(* Logix 5000 project; controller VET 1756-L62 rev 19.52; software revision 19.01; part 24 of 27 *)
(* tags used below, declared in another part *)
   Automatismos : DINT;
   Aux : DINT[500];
   EColor : DINT[1000];
   Eqp : Equipo[50];
   Errors : Fault_Register;
   I : Index;
   RunStarts : DINT[1000];
   String : STRING[40];
   TabEqp : INT[500];
   _Codes : DINT[500];
   _Eqp : Equipo[800];
   _Eqp_Cfg : Eqp_Cfg[800];
   _Origen : Origen[40];
   _Parametros_F : REAL[30];
   _SS : Soft_Starter[20];
   _Typlgie : Eqp_Typologie[800];   // Process Flow Typologie
   Batch : batch[10];
   borrar : DINT[100];
   corriente : REAL[40];
   fecha_plc : DINT;
   flujometro : flujometro[5];
   hora_plc : DINT;
   peso_tolva : REAL[80];
   Set_Global : DINT[20];
   SetDInt : DINT[500];
   simulacion : BOOL;
   SS_Comun : Soft_Starter;
   SSvar : set_variables;
   TabBin : Bins_Setup;
   Timer : TIMER[500];
   Value : DINT[500];
   vdf : VDFS[20];
   VDFidx : DINT;
(* Main1, continued *)

ROUTINE _Cntrl_Valve   (* ladder *)
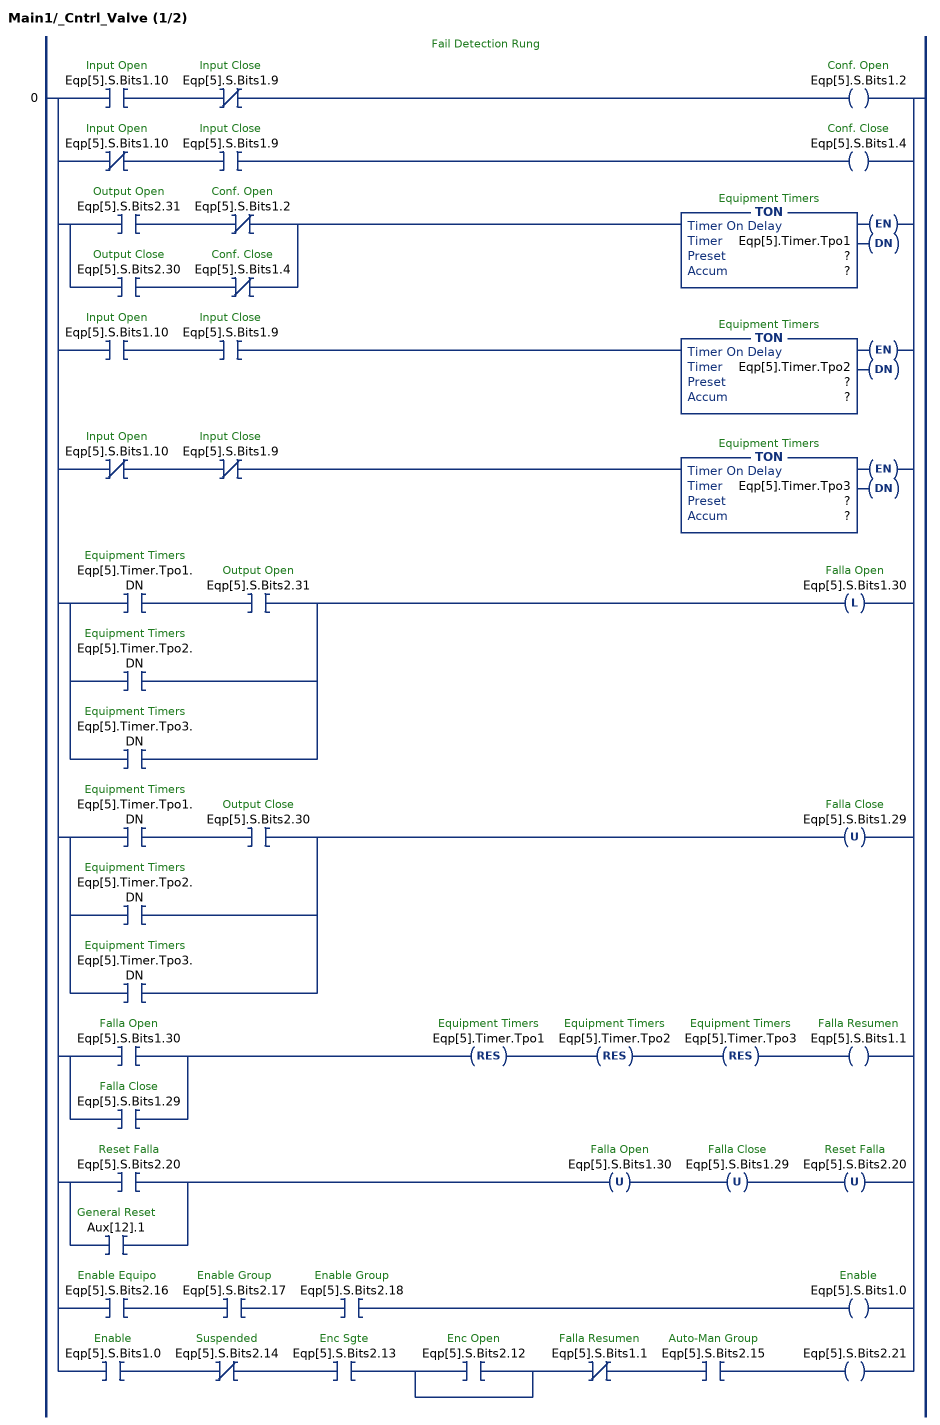
   // Fail Detection Rung
   0: [[XIC(Eqp[5].S.Bits1.10) XIO(Eqp[5].S.Bits1.9) OTE(Eqp[5].S.Bits1.2) ,XIO(Eqp[5].S.Bits1.10) XIC(Eqp[5].S.Bits1.9) OTE(Eqp[5].S.Bits1.4) ] ,[XIC(Eqp[5].S.Bits2.31) XIO(Eqp[5].S.Bits1.2) ,XIC(Eqp[5].S.Bits2.30) XIO(Eqp[5].S.Bits1.4) ] TON(Eqp[5].Timer.Tpo1,?,?) ,XIC(Eqp[5].S.Bits1.10) XIC(Eqp[5].S.Bits1.9) TON(Eqp[5].Timer.Tpo2,?,?) ,XIO(Eqp[5].S.Bits1.10) XIO(Eqp[5].S.Bits1.9) TON(Eqp[5].Timer.Tpo3,?,?) ,[XIC(Eqp[5].Timer.Tpo1.DN) XIC(Eqp[5].S.Bits2.31) ,XIC(Eqp[5].Timer.Tpo2.DN) ,XIC(Eqp[5].Timer.Tpo3.DN) ] OTL(Eqp[5].S.Bits1.30) ,[XIC(Eqp[5].Timer.Tpo1.DN) XIC(Eqp[5].S.Bits2.30) ,XIC(Eqp[5].Timer.Tpo2.DN) ,XIC(Eqp[5].Timer.Tpo3.DN) ] OTU(Eqp[5].S.Bits1.29) ,[XIC(Eqp[5].S.Bits1.30) ,XIC(Eqp[5].S.Bits1.29) ] RES(Eqp[5].Timer.Tpo1) RES(Eqp[5].Timer.Tpo2) RES(Eqp[5].Timer.Tpo3) OTE(Eqp[5].S.Bits1.1) ,[XIC(Eqp[5].S.Bits2.20) ,XIC(Aux[12].1) ] OTU(Eqp[5].S.Bits1.30) OTU(Eqp[5].S.Bits1.29) OTU(Eqp[5].S.Bits2.20) ,XIC(Eqp[5].S.Bits2.16) XIC(Eqp[5].S.Bits2.17) XIC(Eqp[5].S.Bits2.18) OTE(Eqp[5].S.Bits1.0) ,XIC(Eqp[5].S.Bits1.0) XIO(Eqp[5].S.Bits2.14) XIC(Eqp[5].S.Bits2.13) [XIC(Eqp[5].S.Bits2.12) ,] XIO(Eqp[5].S.Bits1.1) XIC(Eqp[5].S.Bits2.15) OTE(Eqp[5].S.Bits2.21) ];
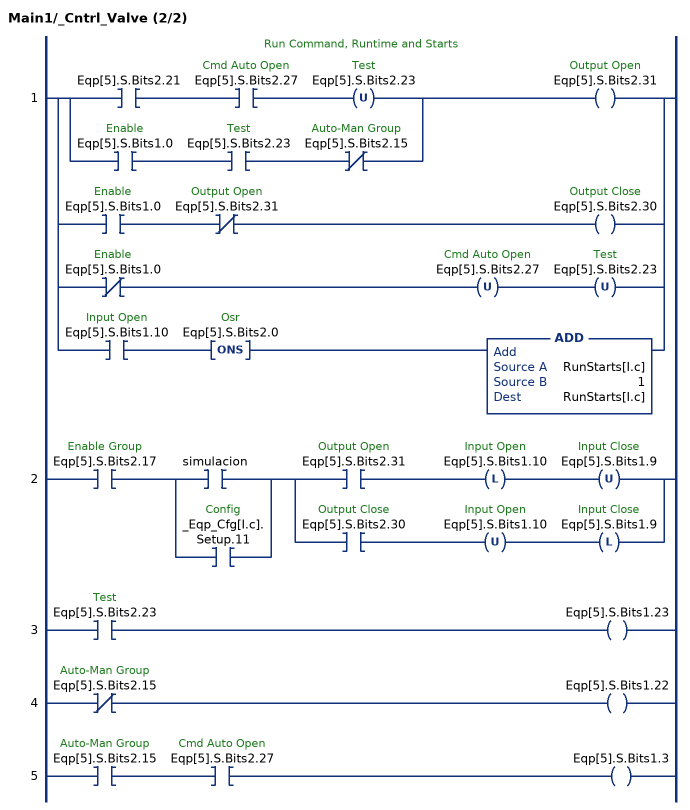
   // Run Command, Runtime and Starts
   1: [[XIC(Eqp[5].S.Bits2.21) XIC(Eqp[5].S.Bits2.27) OTU(Eqp[5].S.Bits2.23) ,XIC(Eqp[5].S.Bits1.0) XIC(Eqp[5].S.Bits2.23) XIO(Eqp[5].S.Bits2.15) ] OTE(Eqp[5].S.Bits2.31) ,XIC(Eqp[5].S.Bits1.0) XIO(Eqp[5].S.Bits2.31) OTE(Eqp[5].S.Bits2.30) ,XIO(Eqp[5].S.Bits1.0) OTU(Eqp[5].S.Bits2.27) OTU(Eqp[5].S.Bits2.23) ,XIC(Eqp[5].S.Bits1.10) ONS(Eqp[5].S.Bits2.0) ADD(RunStarts[I.c],1,RunStarts[I.c]) ];
   2: XIC(Eqp[5].S.Bits2.17)[XIC(simulacion) ,XIC(_Eqp_Cfg[I.c].Setup.11) ][XIC(Eqp[5].S.Bits2.31) OTL(Eqp[5].S.Bits1.10) OTU(Eqp[5].S.Bits1.9) ,XIC(Eqp[5].S.Bits2.30) OTU(Eqp[5].S.Bits1.10) OTL(Eqp[5].S.Bits1.9) ];
   3: XIC(Eqp[5].S.Bits2.23)OTE(Eqp[5].S.Bits1.23);
   4: XIO(Eqp[5].S.Bits2.15)OTE(Eqp[5].S.Bits1.22);
   5: XIC(Eqp[5].S.Bits2.15)XIC(Eqp[5].S.Bits2.27)OTE(Eqp[5].S.Bits1.3);
END_ROUTINE

ROUTINE _Ctrl_SS   (* ladder *)
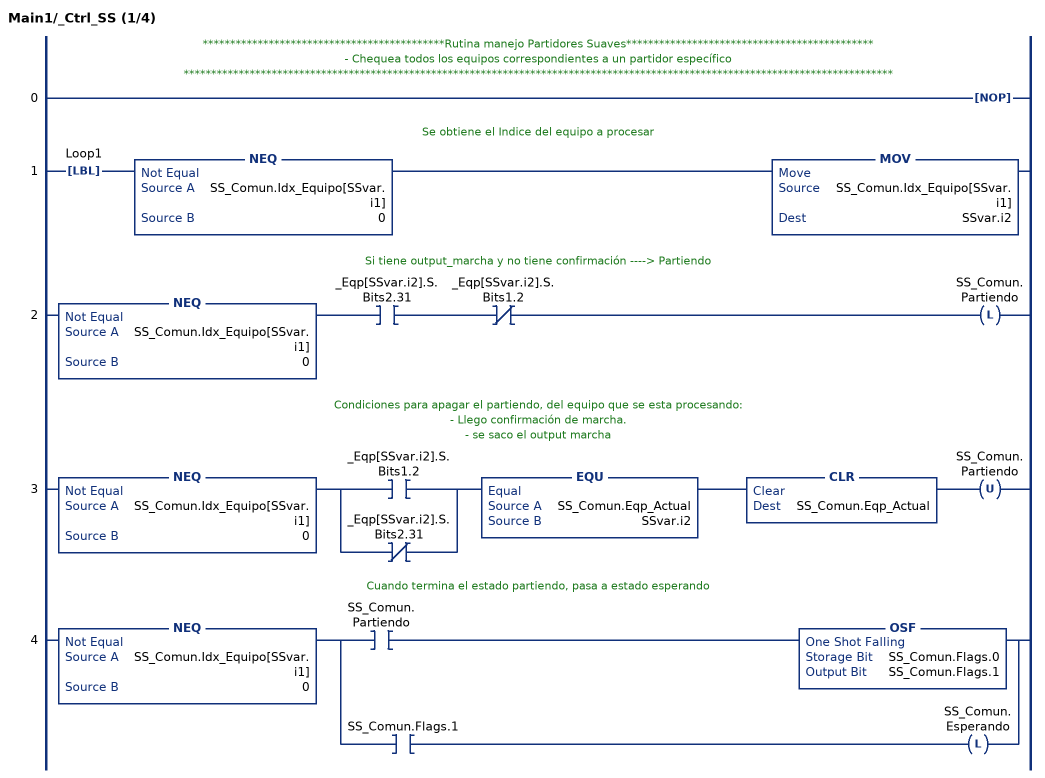
   // ********************************************Rutina manejo Partidores Suaves*********************************************
   // - Chequea todos los equipos correspondientes a un partidor específico
   // *********************************************************************************************************************************
   0: NOP();
   // Se obtiene el Indice del equipo a procesar
   1: LBL(Loop1)NEQ(SS_Comun.Idx_Equipo[SSvar.i1],0)MOV(SS_Comun.Idx_Equipo[SSvar.i1],SSvar.i2);
   // Si tiene output_marcha y no tiene confirmación ----> Partiendo
   2: NEQ(SS_Comun.Idx_Equipo[SSvar.i1],0)XIC(_Eqp[SSvar.i2].S.Bits2.31)XIO(_Eqp[SSvar.i2].S.Bits1.2)OTL(SS_Comun.Partiendo);
   // Condiciones para apagar el partiendo, del equipo que se esta procesando:
   // - Llego confirmación de marcha.
   // - se saco el output marcha
   3: NEQ(SS_Comun.Idx_Equipo[SSvar.i1],0)[XIC(_Eqp[SSvar.i2].S.Bits1.2) ,XIO(_Eqp[SSvar.i2].S.Bits2.31) ]EQU(SS_Comun.Eqp_Actual,SSvar.i2)CLR(SS_Comun.Eqp_Actual)OTU(SS_Comun.Partiendo);
   // Cuando termina el estado partiendo, pasa a estado esperando
   4: NEQ(SS_Comun.Idx_Equipo[SSvar.i1],0)[XIC(SS_Comun.Partiendo) OSF(SS_Comun.Flags.0,SS_Comun.Flags.1) ,XIC(SS_Comun.Flags.1) OTL(SS_Comun.Esperando) ];
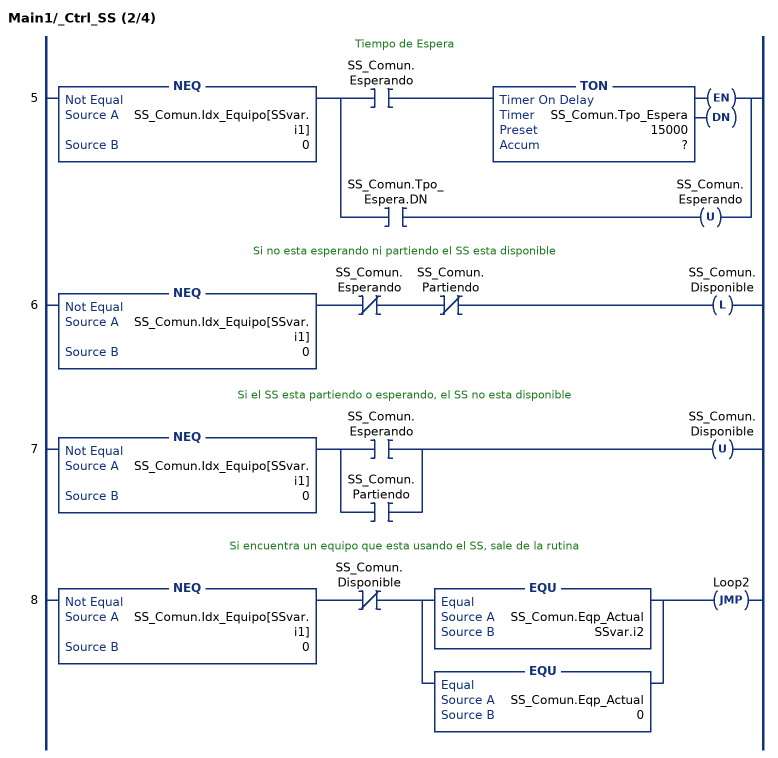
   // Tiempo de Espera
   5: NEQ(SS_Comun.Idx_Equipo[SSvar.i1],0)[XIC(SS_Comun.Esperando) TON(SS_Comun.Tpo_Espera,?,?) ,XIC(SS_Comun.Tpo_Espera.DN) OTU(SS_Comun.Esperando) ];
   // Si no esta esperando ni partiendo el SS esta disponible
   6: NEQ(SS_Comun.Idx_Equipo[SSvar.i1],0)XIO(SS_Comun.Esperando)XIO(SS_Comun.Partiendo)OTL(SS_Comun.Disponible);
   // Si el SS esta partiendo o esperando, el SS no esta disponible
   7: NEQ(SS_Comun.Idx_Equipo[SSvar.i1],0)[XIC(SS_Comun.Esperando) ,XIC(SS_Comun.Partiendo) ]OTU(SS_Comun.Disponible);
   // Si encuentra un equipo que esta usando el SS, sale de la rutina
   8: NEQ(SS_Comun.Idx_Equipo[SSvar.i1],0)XIO(SS_Comun.Disponible)[EQU(SS_Comun.Eqp_Actual,SSvar.i2) ,EQU(SS_Comun.Eqp_Actual,0) ]JMP(Loop2);
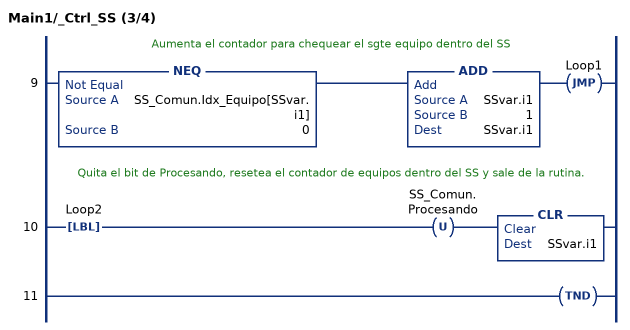
   // Aumenta el contador para chequear el sgte equipo dentro del SS
   9: NEQ(SS_Comun.Idx_Equipo[SSvar.i1],0)ADD(SSvar.i1,1,SSvar.i1)JMP(Loop1);
   // Quita el bit de Procesando, resetea el contador de equipos dentro del SS y sale de la rutina.
   10: LBL(Loop2)OTU(SS_Comun.Procesando)CLR(SSvar.i1);
   11: TND();
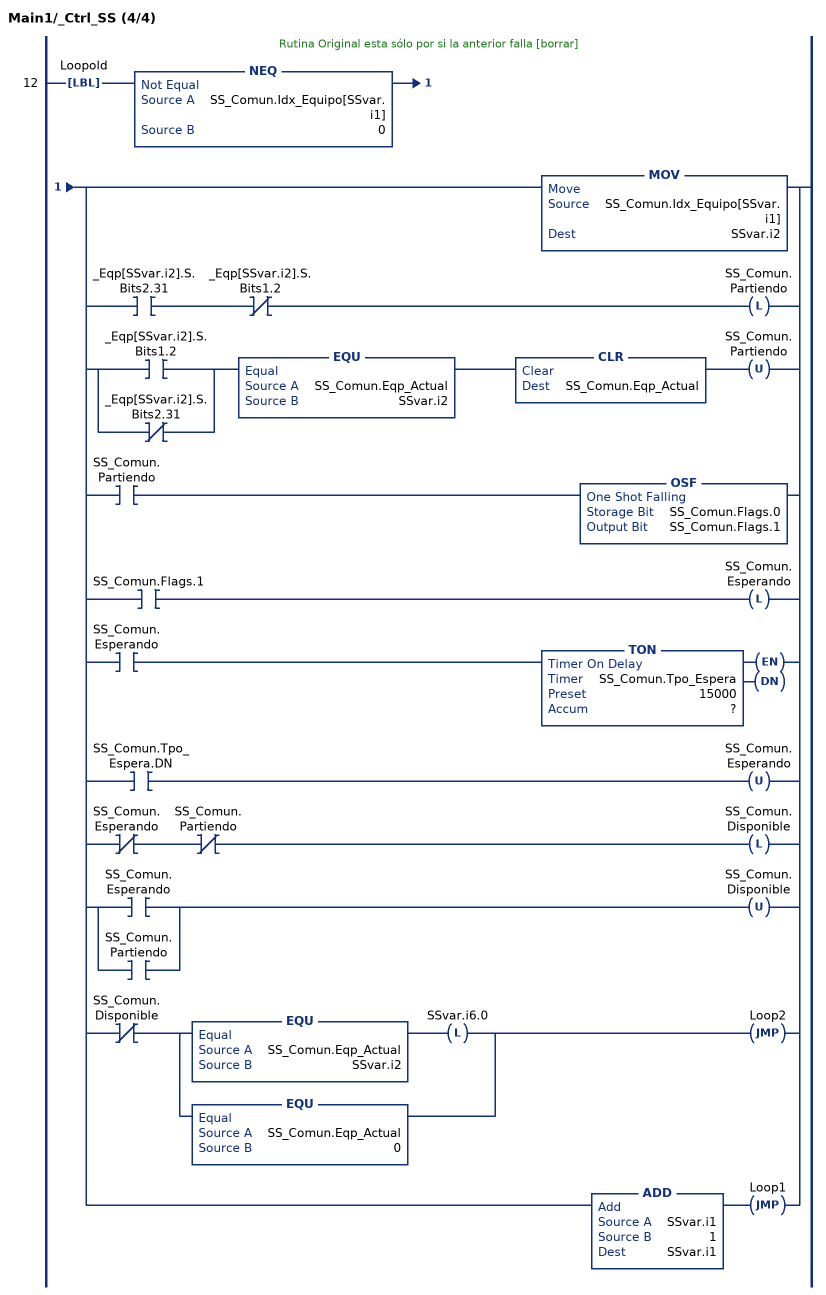
   // Rutina Original esta sólo por si la anterior falla [borrar]
   12: LBL(Loopold)NEQ(SS_Comun.Idx_Equipo[SSvar.i1],0)[[MOV(SS_Comun.Idx_Equipo[SSvar.i1],SSvar.i2) ,XIC(_Eqp[SSvar.i2].S.Bits2.31) XIO(_Eqp[SSvar.i2].S.Bits1.2) OTL(SS_Comun.Partiendo) ,[XIC(_Eqp[SSvar.i2].S.Bits1.2) ,XIO(_Eqp[SSvar.i2].S.Bits2.31) ] EQU(SS_Comun.Eqp_Actual,SSvar.i2) CLR(SS_Comun.Eqp_Actual) OTU(SS_Comun.Partiendo) ,XIC(SS_Comun.Partiendo) OSF(SS_Comun.Flags.0,SS_Comun.Flags.1) ,XIC(SS_Comun.Flags.1) OTL(SS_Comun.Esperando) ,[XIC(SS_Comun.Esperando) TON(SS_Comun.Tpo_Espera,?,?) ,XIC(SS_Comun.Tpo_Espera.DN) OTU(SS_Comun.Esperando) ] ,XIO(SS_Comun.Esperando) XIO(SS_Comun.Partiendo) OTL(SS_Comun.Disponible) ,[XIC(SS_Comun.Esperando) ,XIC(SS_Comun.Partiendo) ] OTU(SS_Comun.Disponible) ,XIO(SS_Comun.Disponible) [EQU(SS_Comun.Eqp_Actual,SSvar.i2) OTL(SSvar.i6.0) ,EQU(SS_Comun.Eqp_Actual,0) ] JMP(Loop2) ] ,ADD(SSvar.i1,1,SSvar.i1) JMP(Loop1) ];
END_ROUTINE

ROUTINE _Ctrl_VDF   (* ladder *)
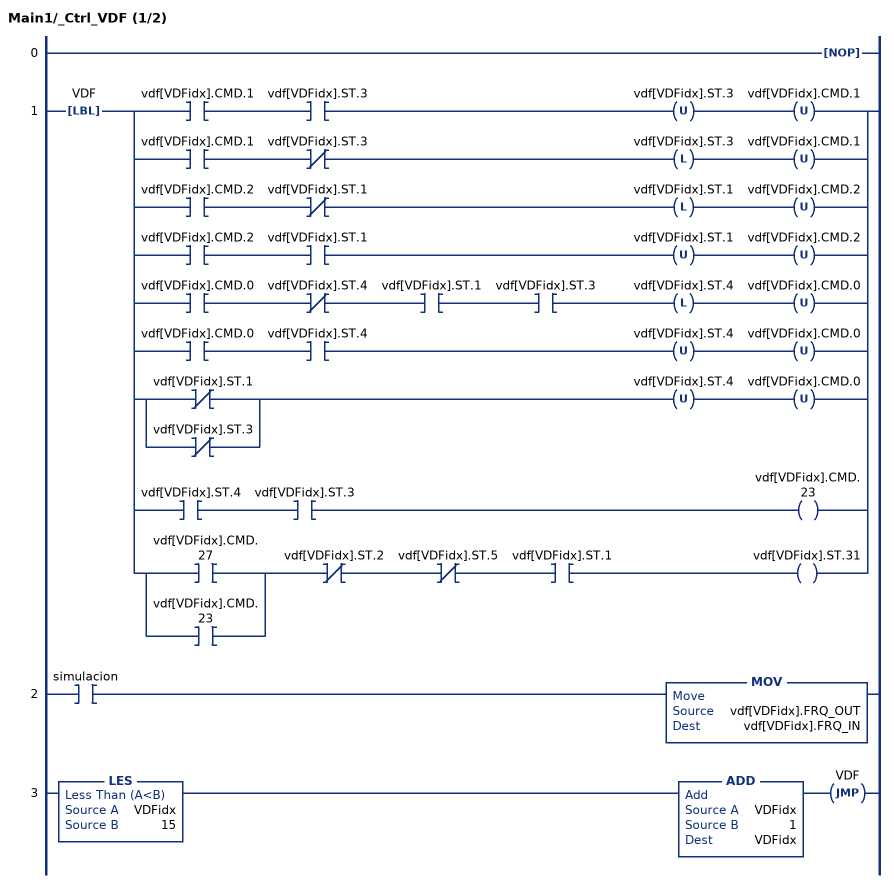
   0: NOP();
   1: LBL(VDF)[XIC(vdf[VDFidx].CMD.1) XIC(vdf[VDFidx].ST.3) OTU(vdf[VDFidx].ST.3) OTU(vdf[VDFidx].CMD.1) ,XIC(vdf[VDFidx].CMD.1) XIO(vdf[VDFidx].ST.3) OTL(vdf[VDFidx].ST.3) OTU(vdf[VDFidx].CMD.1) ,XIC(vdf[VDFidx].CMD.2) XIO(vdf[VDFidx].ST.1) OTL(vdf[VDFidx].ST.1) OTU(vdf[VDFidx].CMD.2) ,XIC(vdf[VDFidx].CMD.2) XIC(vdf[VDFidx].ST.1) OTU(vdf[VDFidx].ST.1) OTU(vdf[VDFidx].CMD.2) ,XIC(vdf[VDFidx].CMD.0) XIO(vdf[VDFidx].ST.4) XIC(vdf[VDFidx].ST.1) XIC(vdf[VDFidx].ST.3) OTL(vdf[VDFidx].ST.4) OTU(vdf[VDFidx].CMD.0) ,XIC(vdf[VDFidx].CMD.0) XIC(vdf[VDFidx].ST.4) OTU(vdf[VDFidx].ST.4) OTU(vdf[VDFidx].CMD.0) ,[XIO(vdf[VDFidx].ST.1) ,XIO(vdf[VDFidx].ST.3) ] OTU(vdf[VDFidx].ST.4) OTU(vdf[VDFidx].CMD.0) ,XIC(vdf[VDFidx].ST.4) XIC(vdf[VDFidx].ST.3) OTE(vdf[VDFidx].CMD.23) ,[XIC(vdf[VDFidx].CMD.27) ,XIC(vdf[VDFidx].CMD.23) ] XIO(vdf[VDFidx].ST.2) XIO(vdf[VDFidx].ST.5) XIC(vdf[VDFidx].ST.1) OTE(vdf[VDFidx].ST.31) ];
   2: XIC(simulacion)MOV(vdf[VDFidx].FRQ_OUT,vdf[VDFidx].FRQ_IN);
   3: LES(VDFidx,15)ADD(VDFidx,1,VDFidx)JMP(VDF);
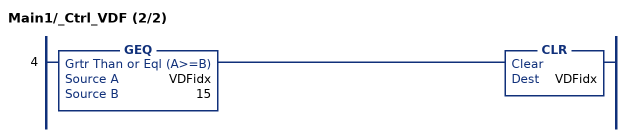
   4: GEQ(VDFidx,15)CLR(VDFidx);
END_ROUTINE

ROUTINE Automatismos_Compuertas_Micros   (* ladder *)
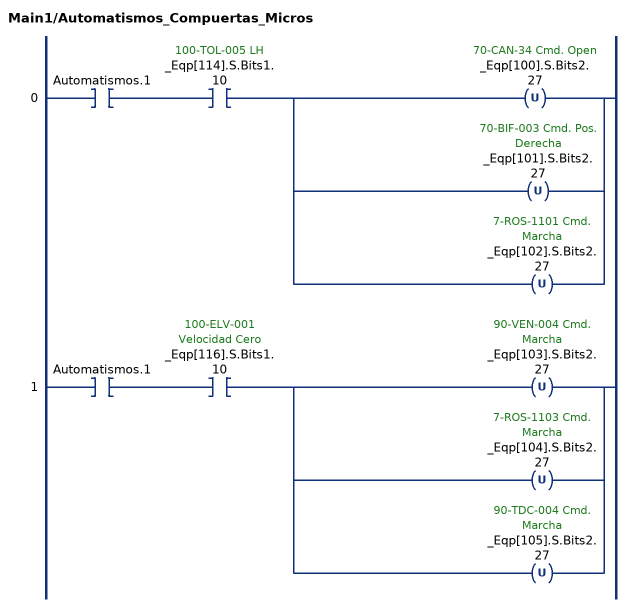
   0: XIC(Automatismos.1)XIC(_Eqp[114].S.Bits1.10)[OTU(_Eqp[100].S.Bits2.27) ,OTU(_Eqp[101].S.Bits2.27) ,OTU(_Eqp[102].S.Bits2.27) ];
   1: XIC(Automatismos.1)XIC(_Eqp[116].S.Bits1.10)[OTU(_Eqp[103].S.Bits2.27) ,OTU(_Eqp[104].S.Bits2.27) ,OTU(_Eqp[105].S.Bits2.27) ];
END_ROUTINE

ROUTINE Automatismos_Filtros   (* ladder *)
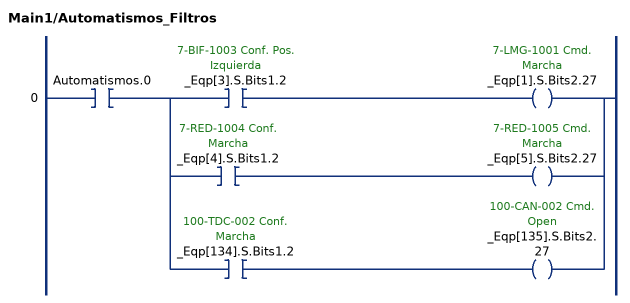
   0: XIC(Automatismos.0)[XIC(_Eqp[3].S.Bits1.2) OTE(_Eqp[1].S.Bits2.27) ,XIC(_Eqp[4].S.Bits1.2) OTE(_Eqp[5].S.Bits2.27) ,XIC(_Eqp[134].S.Bits1.2) OTE(_Eqp[135].S.Bits2.27) ];
END_ROUTINE

ROUTINE Automatismos_valvulas_silos   (* ladder *)
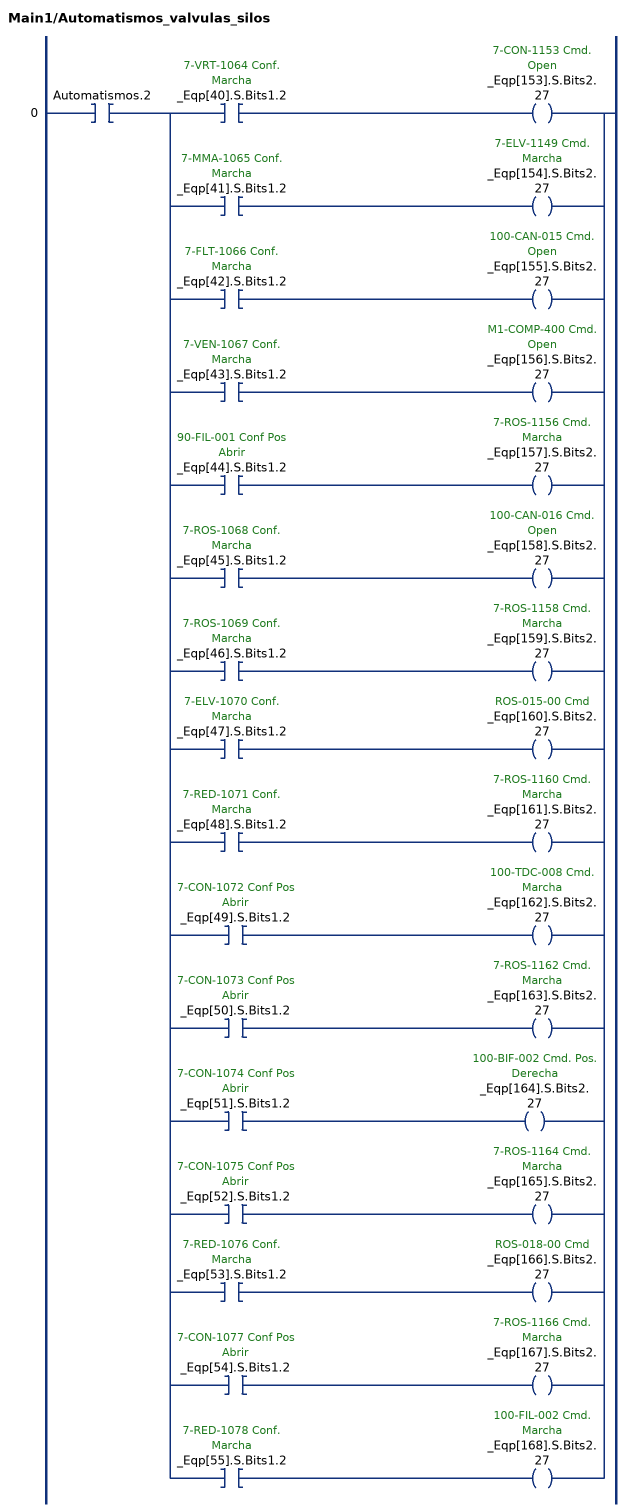
   0: XIC(Automatismos.2)[XIC(_Eqp[40].S.Bits1.2) OTE(_Eqp[153].S.Bits2.27) ,XIC(_Eqp[41].S.Bits1.2) OTE(_Eqp[154].S.Bits2.27) ,XIC(_Eqp[42].S.Bits1.2) OTE(_Eqp[155].S.Bits2.27) ,XIC(_Eqp[43].S.Bits1.2) OTE(_Eqp[156].S.Bits2.27) ,XIC(_Eqp[44].S.Bits1.2) OTE(_Eqp[157].S.Bits2.27) ,XIC(_Eqp[45].S.Bits1.2) OTE(_Eqp[158].S.Bits2.27) ,XIC(_Eqp[46].S.Bits1.2) OTE(_Eqp[159].S.Bits2.27) ,XIC(_Eqp[47].S.Bits1.2) OTE(_Eqp[160].S.Bits2.27) ,XIC(_Eqp[48].S.Bits1.2) OTE(_Eqp[161].S.Bits2.27) ,XIC(_Eqp[49].S.Bits1.2) OTE(_Eqp[162].S.Bits2.27) ,XIC(_Eqp[50].S.Bits1.2) OTE(_Eqp[163].S.Bits2.27) ,XIC(_Eqp[51].S.Bits1.2) OTE(_Eqp[164].S.Bits2.27) ,XIC(_Eqp[52].S.Bits1.2) OTE(_Eqp[165].S.Bits2.27) ,XIC(_Eqp[53].S.Bits1.2) OTE(_Eqp[166].S.Bits2.27) ,XIC(_Eqp[54].S.Bits1.2) OTE(_Eqp[167].S.Bits2.27) ,XIC(_Eqp[55].S.Bits1.2) OTE(_Eqp[168].S.Bits2.27) ];
END_ROUTINE

ROUTINE Codigos   (* ladder *)
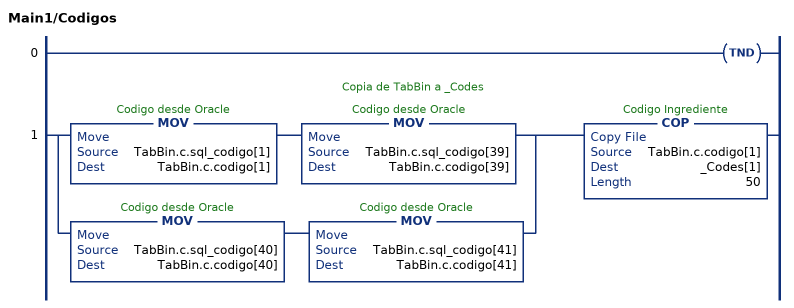
   0: TND();
   // Copia de TabBin a _Codes
   1: [MOV(TabBin.c.sql_codigo[1],TabBin.c.codigo[1]) MOV(TabBin.c.sql_codigo[39],TabBin.c.codigo[39]) ,MOV(TabBin.c.sql_codigo[40],TabBin.c.codigo[40]) MOV(TabBin.c.sql_codigo[41],TabBin.c.codigo[41]) ]COP(TabBin.c.codigo[1],_Codes[1],50);
END_ROUTINE

ROUTINE Enclavamientos   (* ladder *)
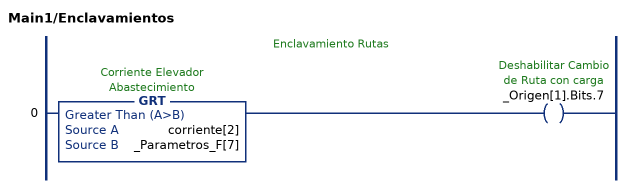
   // Enclavamiento Rutas
   0: GRT(corriente[2],_Parametros_F[7])OTE(_Origen[1].Bits.7);
END_ROUTINE

ROUTINE Error_Handler   (* ladder *)
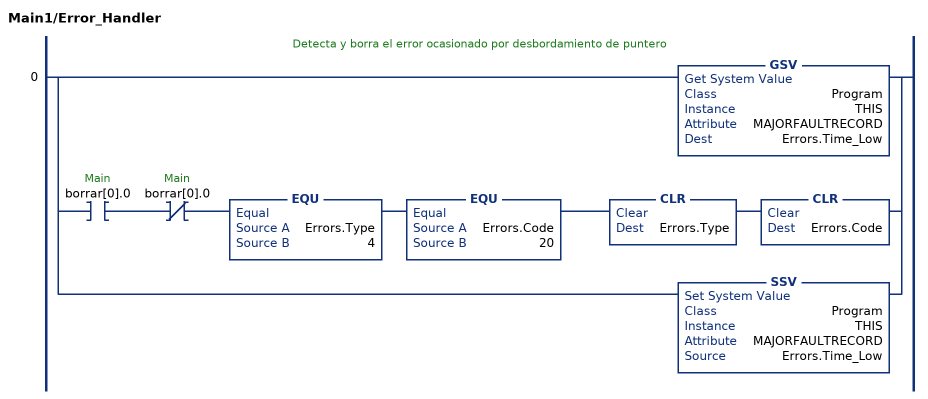
   // Detecta y borra el error ocasionado por desbordamiento de puntero
   0: [GSV(Program,THIS,MAJORFAULTRECORD,Errors.Time_Low) ,XIC(borrar[0].0) XIO(borrar[0].0) EQU(Errors.Type,4) EQU(Errors.Code,20) CLR(Errors.Type) CLR(Errors.Code) ,SSV(Program,THIS,MAJORFAULTRECORD,Errors.Time_Low) ];
END_ROUTINE

ROUTINE Gestion_Flujometros   (* ladder *)
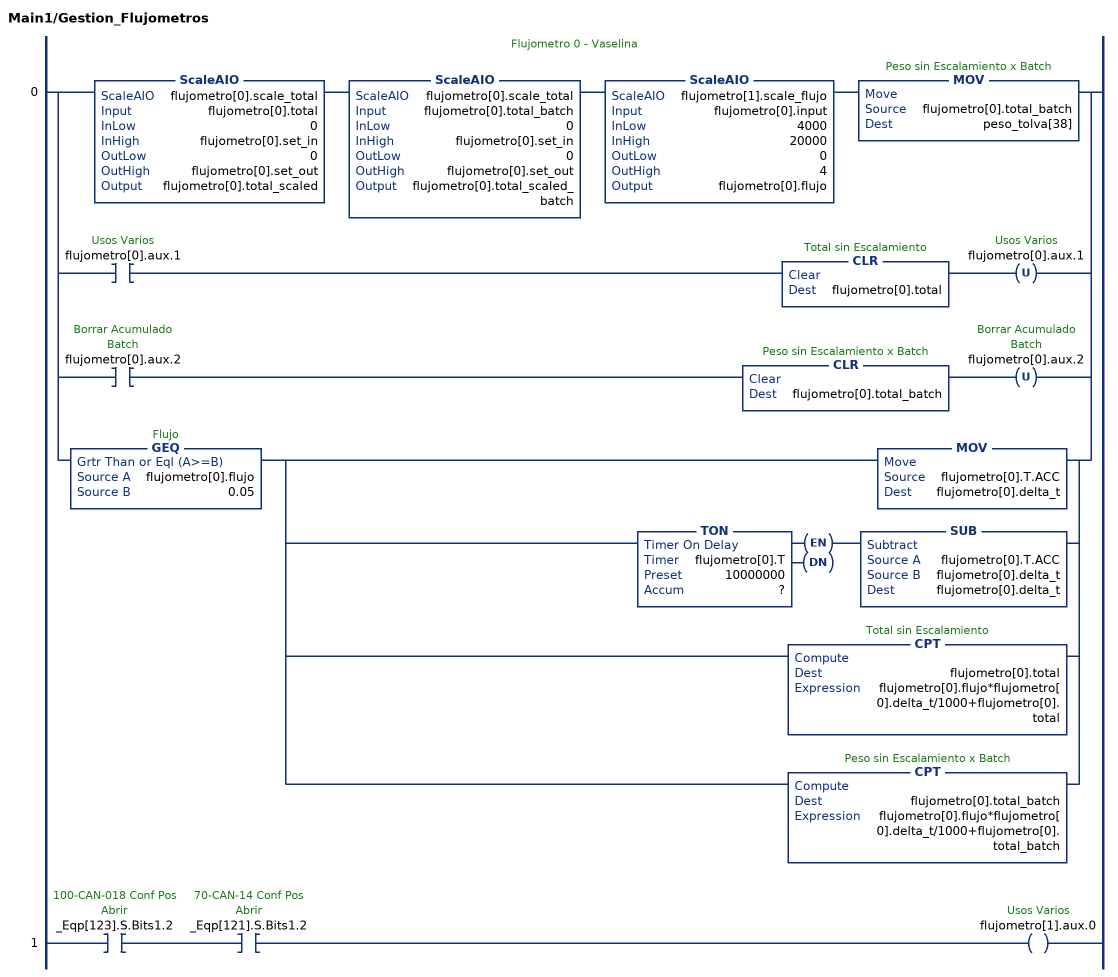
   // Flujometro 0 - Vaselina
   0: [ScaleAIO(flujometro[0].scale_total,flujometro[0].total,0,flujometro[0].set_in,0,flujometro[0].set_out,flujometro[0].total_scaled) ScaleAIO(flujometro[0].scale_total,flujometro[0].total_batch,0,flujometro[0].set_in,0,flujometro[0].set_out,flujometro[0].total_scaled_batch) ScaleAIO(flujometro[1].scale_flujo,flujometro[0].input,4000,20000,0,4,flujometro[0].flujo) MOV(flujometro[0].total_batch,peso_tolva[38]) ,XIC(flujometro[0].aux.1) CLR(flujometro[0].total) OTU(flujometro[0].aux.1) ,XIC(flujometro[0].aux.2) CLR(flujometro[0].total_batch) OTU(flujometro[0].aux.2) ,GEQ(flujometro[0].flujo,0.05) [[MOV(flujometro[0].T.ACC,flujometro[0].delta_t) ,TON(flujometro[0].T,?,?) SUB(flujometro[0].T.ACC,flujometro[0].delta_t,flujometro[0].delta_t) ] ,[CPT(flujometro[0].total,flujometro[0].flujo*flujometro[0].delta_t/1000+flujometro[0].total) ,CPT(flujometro[0].total_batch,flujometro[0].flujo*flujometro[0].delta_t/1000+flujometro[0].total_batch) ] ] ];
   1: XIC(_Eqp[123].S.Bits1.2)XIC(_Eqp[121].S.Bits1.2)OTE(flujometro[1].aux.0);
END_ROUTINE

ROUTINE Main   (* ladder *)
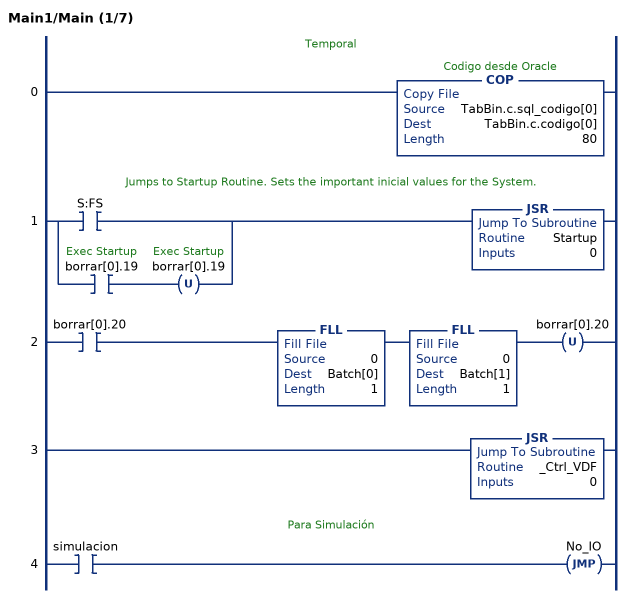
   // Temporal
   0: COP(TabBin.c.sql_codigo[0],TabBin.c.codigo[0],80);
   // Jumps to Startup Routine. Sets the important inicial values for the System.
   1: [XIC(S:FS) ,XIC(borrar[0].19) OTU(borrar[0].19) ]JSR(Startup,0);
   2: XIC(borrar[0].20)FLL(0,Batch[0],1)FLL(0,Batch[1],1)OTU(borrar[0].20);
   3: JSR(_Ctrl_VDF,0);
   // Para Simulación
   4: XIC(simulacion)JMP(No_IO);
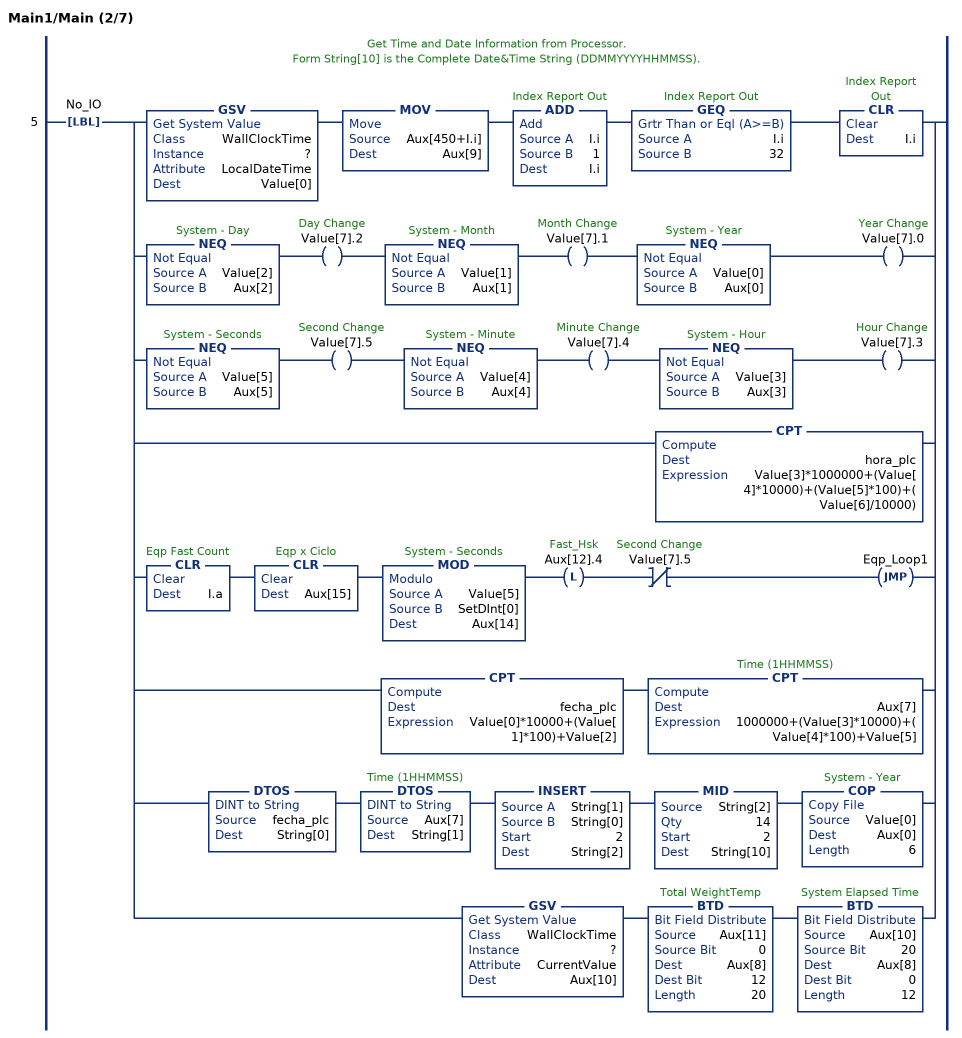
   // Get Time and Date Information from Processor.
   // Form String[10] is the Complete Date&Time String (DDMMYYYYHHMMSS).
   5: LBL(No_IO)[GSV(WallClockTime,?,LocalDateTime,Value[0]) MOV(Aux[450+I.i],Aux[9]) ADD(I.i,1,I.i) GEQ(I.i,32) CLR(I.i) ,NEQ(Value[2],Aux[2]) OTE(Value[7].2) NEQ(Value[1],Aux[1]) OTE(Value[7].1) NEQ(Value[0],Aux[0]) OTE(Value[7].0) ,NEQ(Value[5],Aux[5]) OTE(Value[7].5) NEQ(Value[4],Aux[4]) OTE(Value[7].4) NEQ(Value[3],Aux[3]) OTE(Value[7].3) ,CPT(hora_plc,Value[3]*1000000+(Value[4]*10000)+(Value[5]*100)+(Value[6]/10000)) ,CLR(I.a) CLR(Aux[15]) MOD(Value[5],SetDInt[0],Aux[14]) OTL(Aux[12].4) XIO(Value[7].5) JMP(Eqp_Loop1) ,CPT(fecha_plc,Value[0]*10000+(Value[1]*100)+Value[2]) CPT(Aux[7],1000000+(Value[3]*10000)+(Value[4]*100)+Value[5]) ,DTOS(fecha_plc,String[0]) DTOS(Aux[7],String[1]) INSERT(String[1],String[0],2,String[2]) MID(String[2],14,2,String[10]) COP(Value[0],Aux[0],6) ,GSV(WallClockTime,?,CurrentValue,Aux[10]) BTD(Aux[11],0,Aux[8],12,20) BTD(Aux[10],20,Aux[8],0,12) ];
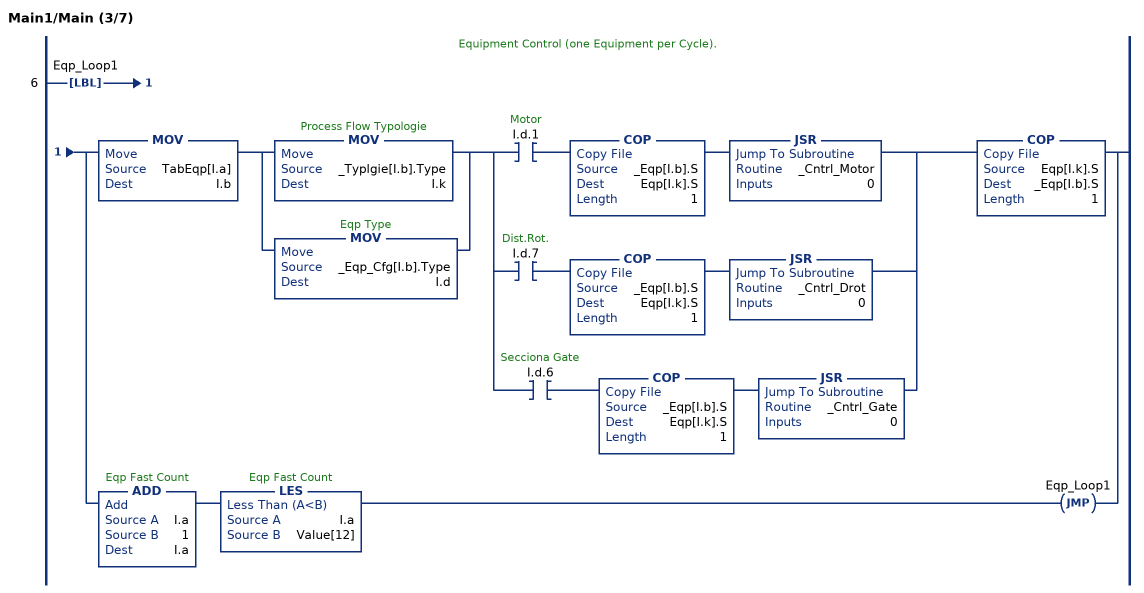
   // Equipment Control (one Equipment per Cycle).
   6: LBL(Eqp_Loop1)[MOV(TabEqp[I.a],I.b) [MOV(_Typlgie[I.b].Type,I.k) ,MOV(_Eqp_Cfg[I.b].Type,I.d) ] [XIC(I.d.1) COP(_Eqp[I.b].S,Eqp[I.k].S,1) JSR(_Cntrl_Motor,0) ,XIC(I.d.7) COP(_Eqp[I.b].S,Eqp[I.k].S,1) JSR(_Cntrl_Drot,0) ,XIC(I.d.6) COP(_Eqp[I.b].S,Eqp[I.k].S,1) JSR(_Cntrl_Gate,0) ] COP(Eqp[I.k].S,_Eqp[I.b].S,1) ,ADD(I.a,1,I.a) LES(I.a,Value[12]) JMP(Eqp_Loop1) ];
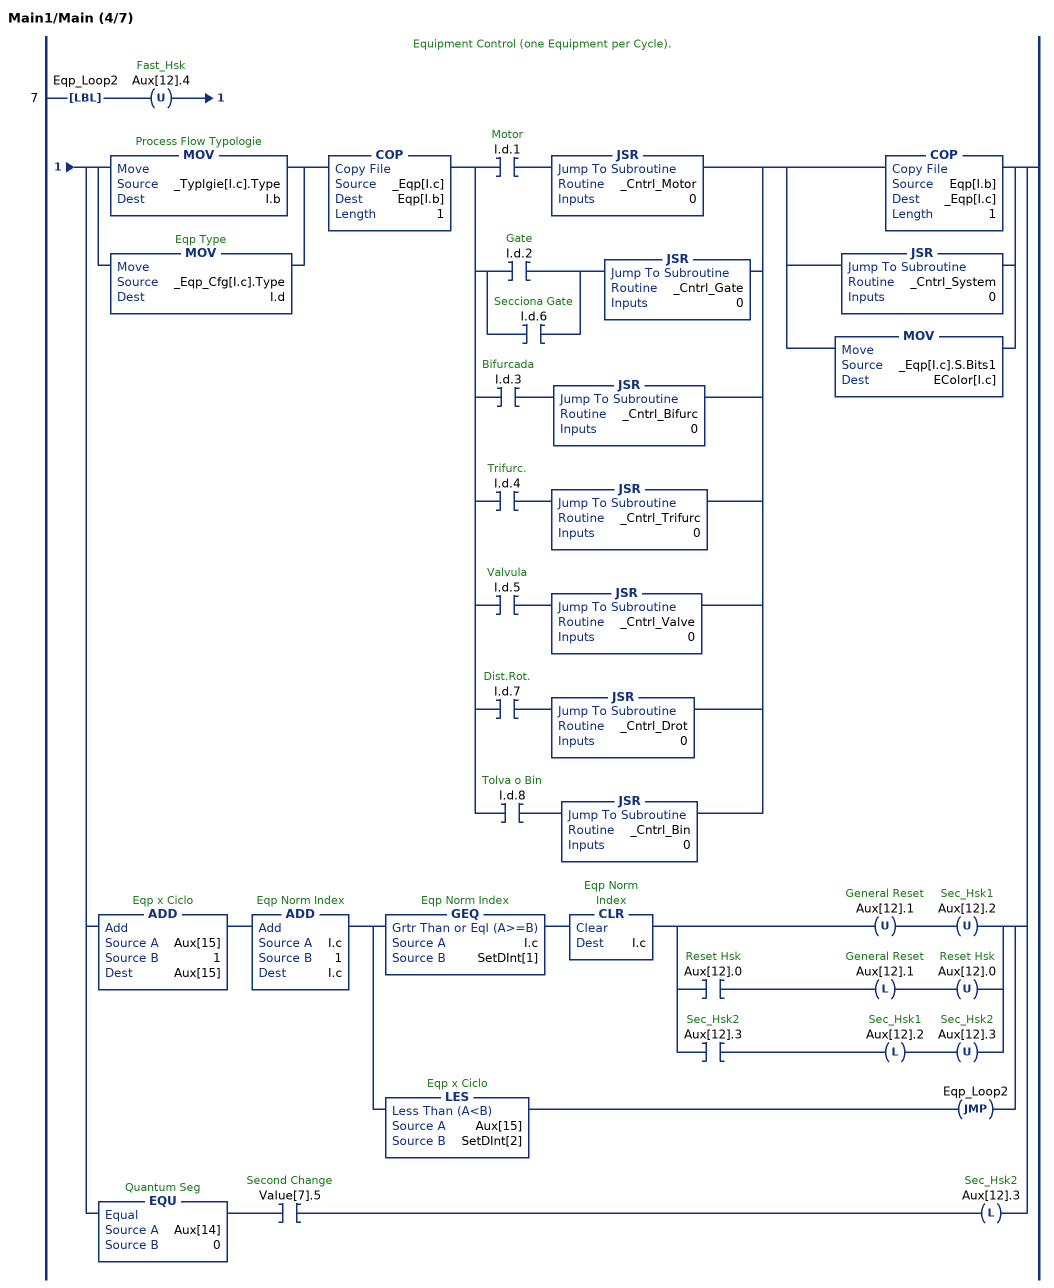
   // Equipment Control (one Equipment per Cycle).
   7: LBL(Eqp_Loop2)OTU(Aux[12].4)[[MOV(_Typlgie[I.c].Type,I.b) ,MOV(_Eqp_Cfg[I.c].Type,I.d) ] COP(_Eqp[I.c],Eqp[I.b],1) [XIC(I.d.1) JSR(_Cntrl_Motor,0) ,[XIC(I.d.2) ,XIC(I.d.6) ] JSR(_Cntrl_Gate,0) ,XIC(I.d.3) JSR(_Cntrl_Bifurc,0) ,XIC(I.d.4) JSR(_Cntrl_Trifurc,0) ,XIC(I.d.5) JSR(_Cntrl_Valve,0) ,XIC(I.d.7) JSR(_Cntrl_Drot,0) ,XIC(I.d.8) JSR(_Cntrl_Bin,0) ] [COP(Eqp[I.b],_Eqp[I.c],1) ,JSR(_Cntrl_System,0) ,MOV(_Eqp[I.c].S.Bits1,EColor[I.c]) ] ,ADD(Aux[15],1,Aux[15]) ADD(I.c,1,I.c) [GEQ(I.c,SetDInt[1]) CLR(I.c) [OTU(Aux[12].1) OTU(Aux[12].2) ,XIC(Aux[12].0) OTL(Aux[12].1) OTU(Aux[12].0) ,XIC(Aux[12].3) OTL(Aux[12].2) OTU(Aux[12].3) ] ,LES(Aux[15],SetDInt[2]) JMP(Eqp_Loop2) ] ,EQU(Aux[14],0) XIC(Value[7].5) OTL(Aux[12].3) ];
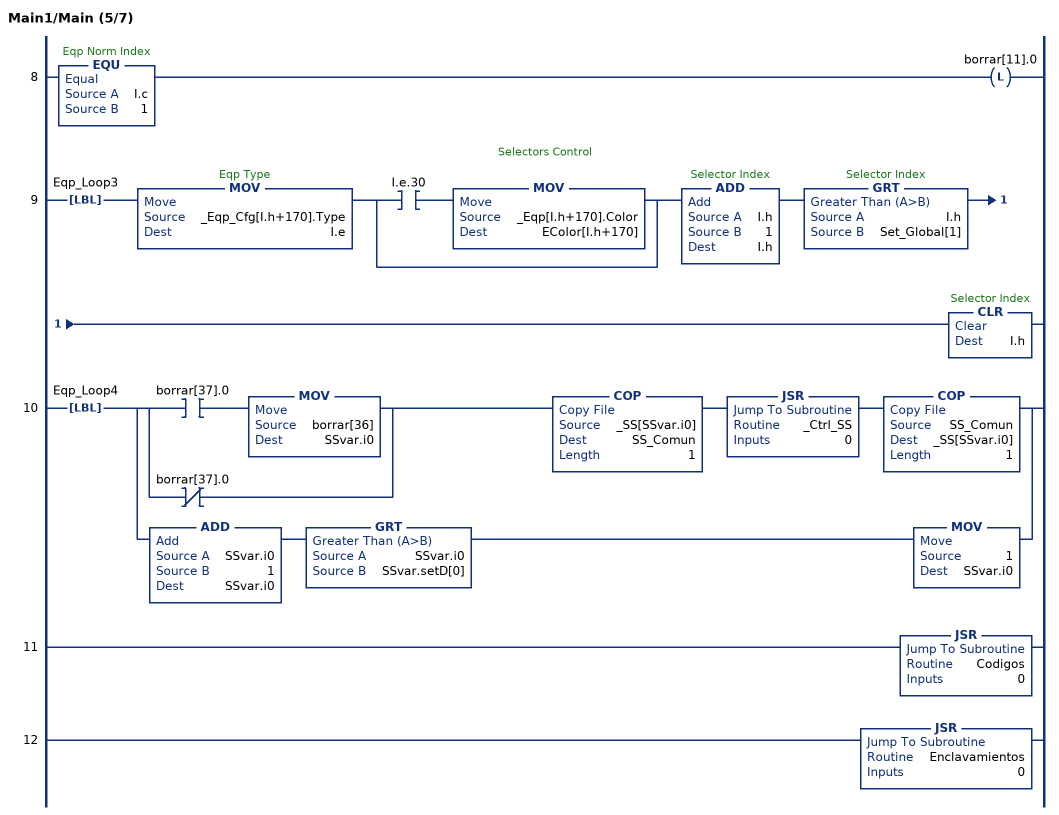
   8: EQU(I.c,1)OTL(borrar[11].0);
   // Selectors Control
   9: LBL(Eqp_Loop3)MOV(_Eqp_Cfg[I.h+170].Type,I.e)[XIC(I.e.30) MOV(_Eqp[I.h+170].Color,EColor[I.h+170]) ,]ADD(I.h,1,I.h)GRT(I.h,Set_Global[1])CLR(I.h);
   10: LBL(Eqp_Loop4)[[XIC(borrar[37].0) MOV(borrar[36],SSvar.i0) ,XIO(borrar[37].0) ] COP(_SS[SSvar.i0],SS_Comun,1) JSR(_Ctrl_SS,0) COP(SS_Comun,_SS[SSvar.i0],1) ,ADD(SSvar.i0,1,SSvar.i0) GRT(SSvar.i0,SSvar.setD[0]) MOV(1,SSvar.i0) ];
   11: JSR(Codigos,0);
   12: JSR(Enclavamientos,0);
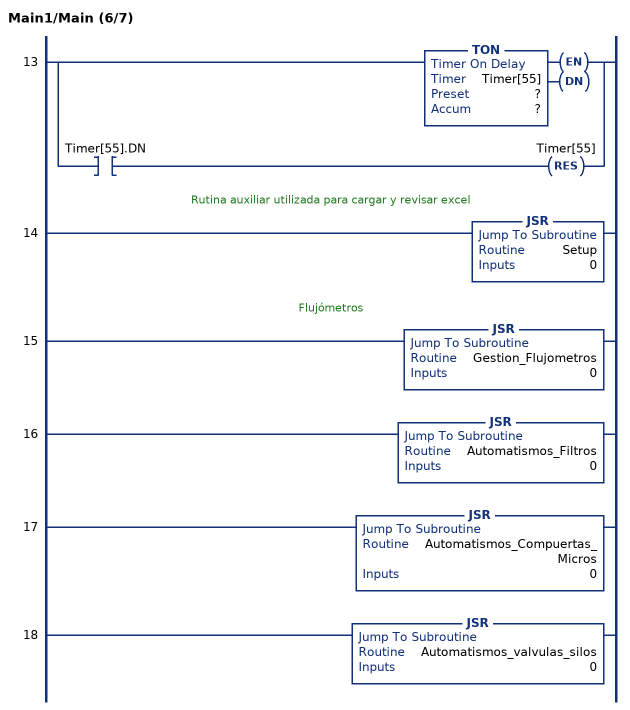
   13: [TON(Timer[55],?,?) ,XIC(Timer[55].DN) RES(Timer[55]) ];
   // Rutina auxiliar utilizada para cargar y revisar excel
   14: JSR(Setup,0);
   // Flujómetros
   15: JSR(Gestion_Flujometros,0);
   16: JSR(Automatismos_Filtros,0);
   17: JSR(Automatismos_Compuertas_Micros,0);
   18: JSR(Automatismos_valvulas_silos,0);
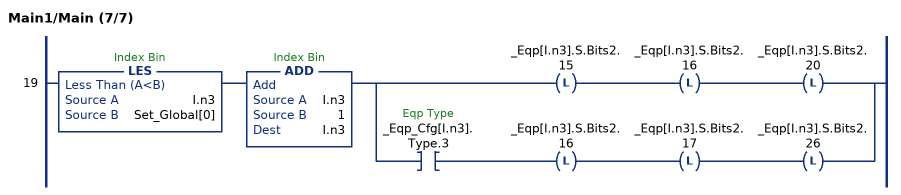
   19: LES(I.n3,Set_Global[0])ADD(I.n3,1,I.n3)[OTL(_Eqp[I.n3].S.Bits2.15) OTL(_Eqp[I.n3].S.Bits2.16) OTL(_Eqp[I.n3].S.Bits2.20) ,XIC(_Eqp_Cfg[I.n3].Type.3) OTL(_Eqp[I.n3].S.Bits2.16) OTL(_Eqp[I.n3].S.Bits2.17) OTL(_Eqp[I.n3].S.Bits2.26) ];
END_ROUTINE
